VAR_GLOBAL

	stLeakTesters							: ST_LeakTester;	
	stHeightTests							: ST_HeightTest;
	stProcessCylinder						: ST_ProcessCylinder;
	stProcessDoor							: ST_ProcessDoor;
	stSlideNest								: ST_SlideNest;
	
END_VAR

(* stored: Version 1.1.0.1, ProductVersion 3.1.4026.18
   GVL GVL_Stations: Id {51987edd-ecbc-463a-bda0-55117182c9fa} *)
